(* CODESYS project Sygnalizacja.project

Project tree, tasks and I/O mapping:
  Device : CODESYS Control Win V3, 3S - Smart Software Solutions GmbH, order no. 305021, version 3.5.8.10
    application Application
      libraries: Standard, * (System)
      task MainTask (cyclic, interval t#20ms, priority 1) calls PLC_PRG
      task VISU_TASK (cyclic, interval 100 ms, priority 31) calls VisuElems.Visu_Prg
      program PLC_PRG [FBD]
      visualisation Visualization
  text list GlobalTextList
*)

// Device/Application/PLC_PRG
PROGRAM PLC_PRG
VAR
	Licznik1: TOF;
	RESET: BOOL;
	CZAS: TIME;
	CZAS_INT: INT;
	CZERWONA_PION: BOOL;
	ZOLTA_PION: BOOL;
	ZIELONA_PION: BOOL;
	Licznik2: TOF;
	CZEKAJ: BOOL;
	CZAS_POZ: TIME;
	CZAS_PION: TIME;
	CZAS_INT_PION: INT;
	CZAS_INT_POZ: INT;
	CZERWONA_POZ: BOOL;
	ZOLTA_POZ: BOOL;
	ZIELONA_POZ: BOOL;
	CZAS_CZEKAJ: TIME;
	CZAS_CZEKAJ_INT: INT;
END_VAR
VAR // added by the converter: edge detectors and wires of the graphical bodies
    _w1, _w2 : BOOL;
END_VAR

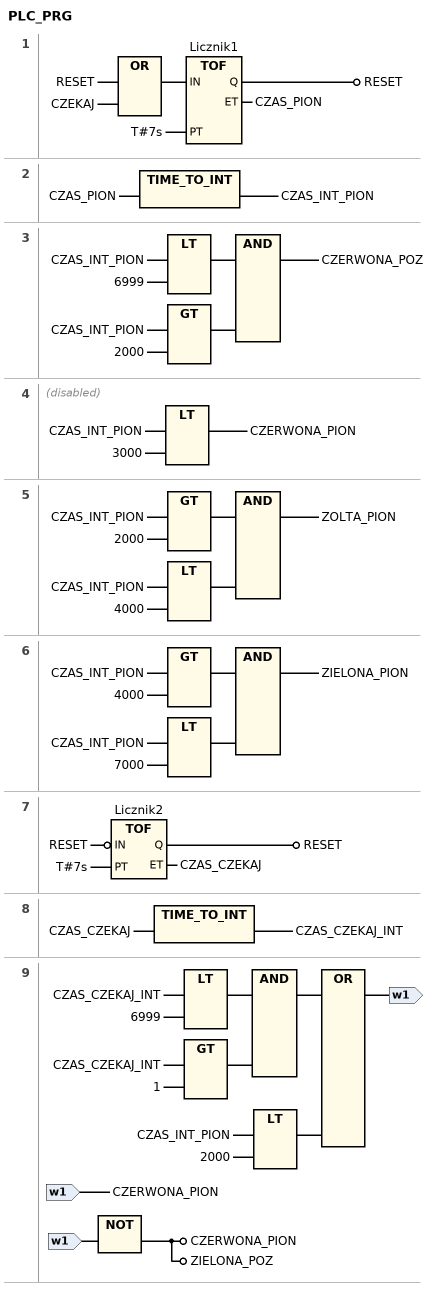
// NETWORK 1
Licznik1(IN := RESET OR CZEKAJ, PT := T#7s, ET => CZAS_PION); // TOF
RESET := NOT Licznik1.Q;

// NETWORK 2
CZAS_INT_PION := TIME_TO_INT(CZAS_PION);

// NETWORK 3
CZERWONA_POZ := CZAS_INT_PION < 6999 AND CZAS_INT_PION > 2000;

// NETWORK 4 (disabled)
// CZERWONA_PION := CZAS_INT_PION < 3000;

// NETWORK 5
ZOLTA_PION := CZAS_INT_PION > 2000 AND CZAS_INT_PION < 4000;

// NETWORK 6
ZIELONA_PION := CZAS_INT_PION > 4000 AND CZAS_INT_PION < 7000;

// NETWORK 7
Licznik2(IN := NOT RESET, PT := T#7s, ET => CZAS_CZEKAJ); // TOF
RESET := NOT Licznik2.Q;

// NETWORK 8
CZAS_CZEKAJ_INT := TIME_TO_INT(CZAS_CZEKAJ);

// NETWORK 9
_w1 := CZAS_CZEKAJ_INT < 6999 AND CZAS_CZEKAJ_INT > 1 OR CZAS_INT_PION < 2000;
CZERWONA_PION := _w1;
_w2 := NOT _w1;
CZERWONA_PION := NOT _w2;
ZIELONA_POZ := NOT _w2;

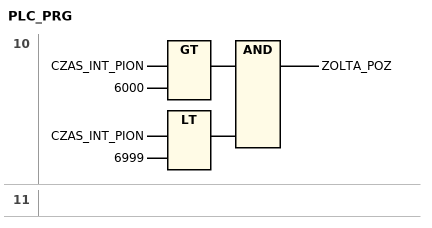
// NETWORK 10
ZOLTA_POZ := CZAS_INT_PION > 6000 AND CZAS_INT_PION < 6999;

// NETWORK 11

END_PROGRAM

// Device/Application/Visualization
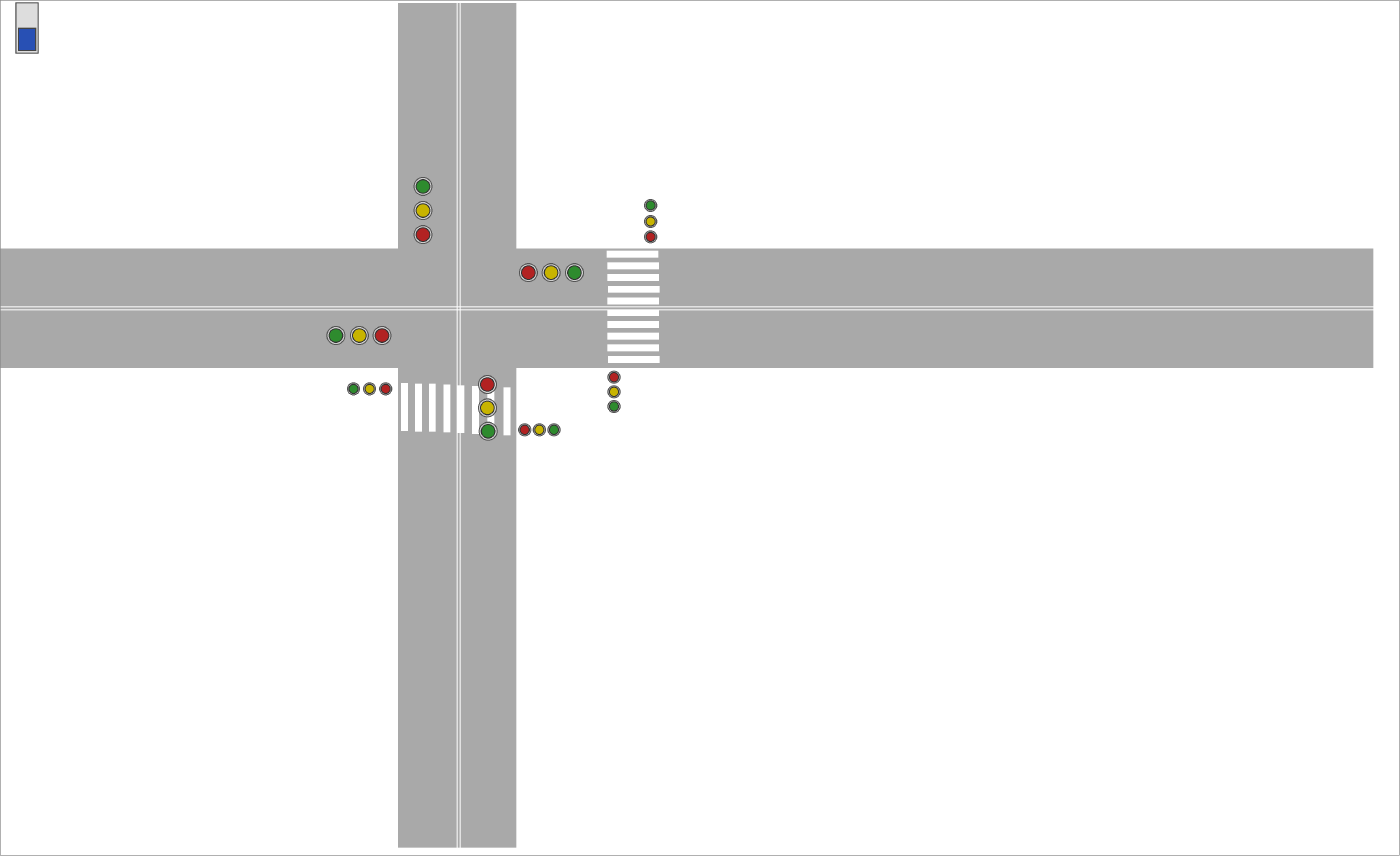
VISUALIZATION Visualization  // 1913x1171
    DipSwitch (2,3 70x70), variable: PLC_PRG.RESET, behaviour: TOGGLE, style: Switch-DipSwitch-Blue
    Rectangle (0,340 544x163)
    Rectangle (544,4 161x1155)
    Rectangle (528,340 1348x163)
    Rectangle (829,343 70x9)
    Rectangle (830,359 70x9)
    Rectangle (830,375 70x9)
    Rectangle (831,391 70x9)
    Rectangle (830,407 70x9)
    Rectangle (830,423 70x9)
    Rectangle (830,439 70x9)
    Rectangle (830,455 70x9)
    Rectangle (830,471 70x9)
    Rectangle (831,487 70x9)
    Rectangle (-3,419 1914x1)
    Rectangle (-6,423 1906x1)
    Rectangle (548,524 9x65)
    Rectangle (567,525 9x65)
    Rectangle (586,525 9x65)
    Rectangle (606,526 9x65)
    Rectangle (625,527 9x65)
    Rectangle (645,528 9x65)
    Rectangle (666,529 9x65)
    Rectangle (688,530 9x65)
    Rectangle (628,2 1x1159)
    Rectangle (624,3 1x1166)
    Lamp1 (563,306 30x30), variable: PLC_PRG.CZERWONA_PION, style: Lamp-Lamp1-Red
    Lamp1 (563,273 30x30), variable: PLC_PRG.ZOLTA_PION, style: Lamp-Lamp1-Yellow
    Lamp1 (563,240 30x30), variable: PLC_PRG.ZIELONA_PION, style: Lamp-Lamp1-Green
    Lamp1 (651,511 30x30), variable: PLC_PRG.CZERWONA_PION, style: Lamp-Lamp1-Red
    Lamp1 (651,543 30x30), variable: PLC_PRG.ZOLTA_PION, style: Lamp-Lamp1-Yellow
    Lamp1 (652,575 30x30), variable: PLC_PRG.ZIELONA_PION, style: Lamp-Lamp1-Green
    Lamp1 (507,444 30x30), variable: PLC_PRG.CZERWONA_POZ, style: Lamp-Lamp1-Red
    Lamp1 (476,444 30x30), variable: PLC_PRG.ZOLTA_POZ, style: Lamp-Lamp1-Yellow
    Lamp1 (444,444 30x30), variable: PLC_PRG.ZIELONA_POZ, style: Lamp-Lamp1-Green
    Lamp1 (707,358 30x30), variable: PLC_PRG.CZERWONA_POZ, style: Lamp-Lamp1-Red
    Lamp1 (738,358 30x30), variable: PLC_PRG.ZOLTA_POZ, style: Lamp-Lamp1-Yellow
    Lamp1 (770,358 30x30), variable: PLC_PRG.ZIELONA_POZ, style: Lamp-Lamp1-Green
    Lamp1 (829,506 20x20), variable: PLC_PRG.CZERWONA_PION, style: Lamp-Lamp1-Red
    Lamp1 (829,526 20x20), variable: PLC_PRG.ZOLTA_PION, style: Lamp-Lamp1-Yellow
    Lamp1 (829,546 20x20), variable: PLC_PRG.ZIELONA_PION, style: Lamp-Lamp1-Green
    Lamp1 (879,314 20x20), variable: PLC_PRG.CZERWONA_PION, style: Lamp-Lamp1-Red
    Lamp1 (879,293 20x20), variable: PLC_PRG.ZOLTA_PION, style: Lamp-Lamp1-Yellow
    Lamp1 (879,271 20x20), variable: PLC_PRG.ZIELONA_PION, style: Lamp-Lamp1-Green
    Lamp1 (707,578 20x20), variable: PLC_PRG.CZERWONA_POZ, style: Lamp-Lamp1-Red
    Lamp1 (727,578 20x20), variable: PLC_PRG.ZOLTA_POZ, style: Lamp-Lamp1-Yellow
    Lamp1 (747,578 20x20), variable: PLC_PRG.ZIELONA_POZ, style: Lamp-Lamp1-Green
    Lamp1 (517,522 20x20), variable: PLC_PRG.CZERWONA_POZ, style: Lamp-Lamp1-Red
    Lamp1 (495,522 20x20), variable: PLC_PRG.ZOLTA_POZ, style: Lamp-Lamp1-Yellow
    Lamp1 (473,522 20x20), variable: PLC_PRG.ZIELONA_POZ, style: Lamp-Lamp1-Green
END_VISUALIZATION
